FUNCTION_BLOCK SignalTower
VAR
	ledRed		: LedLamp;
	ledGreen	: LedLamp;
END_VAR

METHOD SetStateOP
VAR_INPUT
END_VAR
ledRed.Off();
ledGreen.On();
END_METHOD

METHOD SetStateSTOP
VAR_INPUT
END_VAR
ledRed.On();
ledGreen.Off();
END_METHOD

END_FUNCTION_BLOCK

(* stored: Version 1.1.0.1, ProductVersion 3.1.4024.12
   POU SignalTower: Id {1bc1d9f1-4b08-4753-811a-6c0cb149c74c}, SpecialFunc None
   Method SetStateOP: Id {ac0a33a4-85c0-4eb1-b53f-4bfb796657d7}
   Method SetStateSTOP: Id {7ff2222a-d190-4541-bdae-d3f3a35b03b1} *)
